KUKA KRL program: sieben_mit.src, sieben_mit.dat

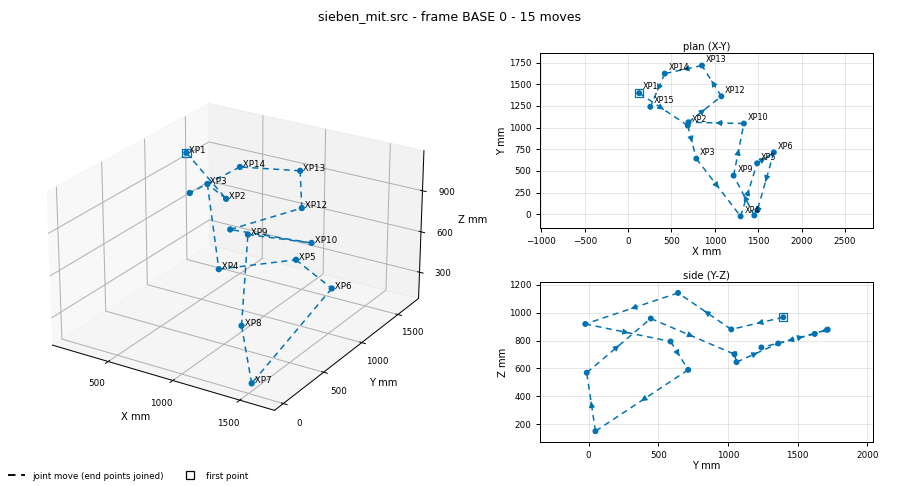
[picture p0: tool path of sieben_mit.src in frame BASE 0, 15 of 17 moves have a stored position in this frame; points joined in program order, loops and branches not executed]
--- sieben_mit.src ---
&ACCESS RVP
&REL 30
&PARAM EDITMASK = *
&PARAM TEMPLATE = C:\KRC\Roboter\Template\vorgabe
DEF sieben_mit( )
;FOLD INI;%{PE}
  ;FOLD BASISTECH INI
    GLOBAL INTERRUPT DECL 3 WHEN $STOPMESS==TRUE DO IR_STOPM ( )
    INTERRUPT ON 3
    BAS (#INITMOV,0 )
  ;ENDFOLD (BASISTECH INI)
  ;FOLD USER INI
    ;Make your modifications here

  ;ENDFOLD (USER INI)
;ENDFOLD (INI)

;FOLD PTP HOME Vel=10 % DEFAULT;%{PE}%R 8.3.40,%MKUKATPBASIS,%CMOVE,%VPTP,%P 1:PTP, 2:HOME, 3:, 5:10, 7:DEFAULT
$BWDSTART=FALSE
PDAT_ACT=PDEFAULT
FDAT_ACT=FHOME
BAS(#PTP_PARAMS,10)
$H_POS=XHOME
PTP XHOME
;ENDFOLD

WAIT FOR IS_KEY_PRESSED(12)

;FOLD PTP P1 Vel=30 % PDAT1 Tool[12]:jan_test Base[0];%{PE}%R 8.3.40,%MKUKATPBASIS,%CMOVE,%VPTP,%P 1:PTP, 2:P1, 3:, 5:30, 7:PDAT1
$BWDSTART=FALSE
PDAT_ACT=PPDAT1
FDAT_ACT=FP1
BAS(#PTP_PARAMS,30)
PTP XP1
;ENDFOLD

WAIT FOR IS_KEY_PRESSED(12)

;FOLD PTP P2 Vel=30 % PDAT2 Tool[12]:jan_test Base[0];%{PE}%R 8.3.40,%MKUKATPBASIS,%CMOVE,%VPTP,%P 1:PTP, 2:P2, 3:, 5:30, 7:PDAT2
$BWDSTART=FALSE
PDAT_ACT=PPDAT2
FDAT_ACT=FP2
BAS(#PTP_PARAMS,30)
PTP XP2
;ENDFOLD

WAIT FOR IS_KEY_PRESSED(12)

;FOLD PTP P3 Vel=30 % PDAT3 Tool[12]:jan_test Base[0];%{PE}%R 8.3.40,%MKUKATPBASIS,%CMOVE,%VPTP,%P 1:PTP, 2:P3, 3:, 5:30, 7:PDAT3
$BWDSTART=FALSE
PDAT_ACT=PPDAT3
FDAT_ACT=FP3
BAS(#PTP_PARAMS,30)
PTP XP3
;ENDFOLD

WAIT FOR IS_KEY_PRESSED(12)

;FOLD PTP P4 Vel=30 % PDAT4 Tool[12]:jan_test Base[0];%{PE}%R 8.3.40,%MKUKATPBASIS,%CMOVE,%VPTP,%P 1:PTP, 2:P4, 3:, 5:30, 7:PDAT4
$BWDSTART=FALSE
PDAT_ACT=PPDAT4
FDAT_ACT=FP4
BAS(#PTP_PARAMS,30)
PTP XP4
;ENDFOLD

WAIT FOR IS_KEY_PRESSED(12)

;FOLD PTP P5 Vel=30 % PDAT5 Tool[12]:jan_test Base[0];%{PE}%R 8.3.40,%MKUKATPBASIS,%CMOVE,%VPTP,%P 1:PTP, 2:P5, 3:, 5:30, 7:PDAT5
$BWDSTART=FALSE
PDAT_ACT=PPDAT5
FDAT_ACT=FP5
BAS(#PTP_PARAMS,30)
PTP XP5
;ENDFOLD

WAIT FOR IS_KEY_PRESSED(12)

;FOLD PTP P6 Vel=30 % PDAT6 Tool[12]:jan_test Base[0];%{PE}%R 8.3.40,%MKUKATPBASIS,%CMOVE,%VPTP,%P 1:PTP, 2:P6, 3:, 5:30, 7:PDAT6
$BWDSTART=FALSE
PDAT_ACT=PPDAT6
FDAT_ACT=FP6
BAS(#PTP_PARAMS,30)
PTP XP6
;ENDFOLD

WAIT FOR IS_KEY_PRESSED(12)

;FOLD PTP P7 Vel=30 % PDAT7 Tool[12]:jan_test Base[0];%{PE}%R 8.3.40,%MKUKATPBASIS,%CMOVE,%VPTP,%P 1:PTP, 2:P7, 3:, 5:30, 7:PDAT7
$BWDSTART=FALSE
PDAT_ACT=PPDAT7
FDAT_ACT=FP7
BAS(#PTP_PARAMS,30)
PTP XP7
;ENDFOLD

WAIT FOR IS_KEY_PRESSED(12)

;FOLD PTP P8 Vel=30 % PDAT8 Tool[12]:jan_test Base[0];%{PE}%R 8.3.40,%MKUKATPBASIS,%CMOVE,%VPTP,%P 1:PTP, 2:P8, 3:, 5:30, 7:PDAT8
$BWDSTART=FALSE
PDAT_ACT=PPDAT8
FDAT_ACT=FP8
BAS(#PTP_PARAMS,30)
PTP XP8
;ENDFOLD

WAIT FOR IS_KEY_PRESSED(12)

;FOLD PTP P9 Vel=30 % PDAT9 Tool[12]:jan_test Base[0];%{PE}%R 8.3.40,%MKUKATPBASIS,%CMOVE,%VPTP,%P 1:PTP, 2:P9, 3:, 5:30, 7:PDAT9
$BWDSTART=FALSE
PDAT_ACT=PPDAT9
FDAT_ACT=FP9
BAS(#PTP_PARAMS,30)
PTP XP9
;ENDFOLD

WAIT FOR IS_KEY_PRESSED(12)

;FOLD PTP P10 Vel=30 % PDAT10 Tool[12]:jan_test Base[0];%{PE}%R 8.3.40,%MKUKATPBASIS,%CMOVE,%VPTP,%P 1:PTP, 2:P10, 3:, 5:30, 7:PDAT10
$BWDSTART=FALSE
PDAT_ACT=PPDAT10
FDAT_ACT=FP10
BAS(#PTP_PARAMS,30)
PTP XP10
;ENDFOLD

WAIT FOR IS_KEY_PRESSED(12)

;FOLD PTP P11 Vel=30 % PDAT11 Tool[12]:jan_test Base[0];%{PE}%R 8.3.40,%MKUKATPBASIS,%CMOVE,%VPTP,%P 1:PTP, 2:P11, 3:, 5:30, 7:PDAT11
$BWDSTART=FALSE
PDAT_ACT=PPDAT11
FDAT_ACT=FP11
BAS(#PTP_PARAMS,30)
PTP XP11
;ENDFOLD

WAIT FOR IS_KEY_PRESSED(12)

;FOLD PTP P12 Vel=30 % PDAT12 Tool[12]:jan_test Base[0];%{PE}%R 8.3.40,%MKUKATPBASIS,%CMOVE,%VPTP,%P 1:PTP, 2:P12, 3:, 5:30, 7:PDAT12
$BWDSTART=FALSE
PDAT_ACT=PPDAT12
FDAT_ACT=FP12
BAS(#PTP_PARAMS,30)
PTP XP12
;ENDFOLD

WAIT FOR IS_KEY_PRESSED(12)

;FOLD PTP P13 Vel=30 % PDAT13 Tool[12]:jan_test Base[0];%{PE}%R 8.3.40,%MKUKATPBASIS,%CMOVE,%VPTP,%P 1:PTP, 2:P13, 3:, 5:30, 7:PDAT13
$BWDSTART=FALSE
PDAT_ACT=PPDAT13
FDAT_ACT=FP13
BAS(#PTP_PARAMS,30)
PTP XP13
;ENDFOLD

WAIT FOR IS_KEY_PRESSED(12)

;FOLD PTP P14 Vel=30 % PDAT14 Tool[12]:jan_test Base[0];%{PE}%R 8.3.40,%MKUKATPBASIS,%CMOVE,%VPTP,%P 1:PTP, 2:P14, 3:, 5:30, 7:PDAT14
$BWDSTART=FALSE
PDAT_ACT=PPDAT14
FDAT_ACT=FP14
BAS(#PTP_PARAMS,30)
PTP XP14
;ENDFOLD

WAIT FOR IS_KEY_PRESSED(12)

;FOLD PTP P15 Vel=30 % PDAT15 Tool[12]:jan_test Base[0];%{PE}%R 8.3.40,%MKUKATPBASIS,%CMOVE,%VPTP,%P 1:PTP, 2:P15, 3:, 5:30, 7:PDAT15
$BWDSTART=FALSE
PDAT_ACT=PPDAT15
FDAT_ACT=FP15
BAS(#PTP_PARAMS,30)
PTP XP15
;ENDFOLD







;FOLD PTP HOME Vel=10 % DEFAULT;%{PE}%R 8.3.40,%MKUKATPBASIS,%CMOVE,%VPTP,%P 1:PTP, 2:HOME, 3:, 5:10, 7:DEFAULT
$BWDSTART=FALSE
PDAT_ACT=PDEFAULT
FDAT_ACT=FHOME
BAS(#PTP_PARAMS,10)
$H_POS=XHOME
PTP XHOME
;ENDFOLD

END

--- sieben_mit.dat ---
&ACCESS RVP
&REL 30
&PARAM EDITMASK = *
&PARAM TEMPLATE = C:\KRC\Roboter\Template\vorgabe
DEFDAT  sieben_mit
;FOLD EXTERNAL DECLARATIONS;%{PE}%MKUKATPBASIS,%CEXT,%VCOMMON,%P
;FOLD BASISTECH EXT;%{PE}%MKUKATPBASIS,%CEXT,%VEXT,%P
EXT  BAS (BAS_COMMAND  :IN,REAL  :IN )
DECL INT SUCCESS
;ENDFOLD (BASISTECH EXT)
;FOLD USER EXT;%{E}%MKUKATPUSER,%CEXT,%VEXT,%P
;Make your modifications here

;ENDFOLD (USER EXT)
;ENDFOLD (EXTERNAL DECLARATIONS)
DECL BASIS_SUGG_T LAST_BASIS={POINT1[] "P15                     ",POINT2[] "P15                     ",CP_PARAMS[] "CPDAT0                  ",PTP_PARAMS[] "PDAT15                  ",CONT[] "                        ",CP_VEL[] "2.0                     ",PTP_VEL[] "30                      ",SYNC_PARAMS[] "SYNCDAT                 ",SPL_NAME[] "S0                      ",A_PARAMS[] "ADAT0                   "}
DECL E6POS XP1={X 127.121788,Y 1397.60730,Z 966.878418,A 28.9919910,B 72.7776489,C -80.1574097,S 18,T 35,E1 0.00499581080,E2 20160.0,E3 0.0,E4 0.0,E5 0.0,E6 0.0}
DECL FDAT FP1={TOOL_NO 12,BASE_NO 0,IPO_FRAME #BASE,POINT2[] " ",TQ_STATE FALSE}
DECL PDAT PPDAT1={VEL 100.000,ACC 50.0000,APO_DIST 100.000,APO_MODE #CDIS,GEAR_JERK 50.0000,EXAX_IGN 0}
DECL E6POS XP2={X 687.482056,Y 1024.24646,Z 879.843384,A 158.221695,B 27.4421253,C 130.372269,S 18,T 35,E1 0.00499581080,E2 20160.0,E3 0.0,E4 0.0,E5 0.0,E6 0.0}
DECL FDAT FP2={TOOL_NO 12,BASE_NO 0,IPO_FRAME #BASE,POINT2[] " ",TQ_STATE FALSE}
DECL PDAT PPDAT2={VEL 100.000,ACC 50.0000,APO_DIST 100.000,APO_MODE #CDIS,GEAR_JERK 50.0000,EXAX_IGN 0}
DECL E6POS XP3={X 786.710938,Y 642.340820,Z 1141.43823,A -17.2900,B 75.0733795,C -84.1357117,S 18,T 35,E1 0.00499581080,E2 20160.0,E3 0.0,E4 0.0,E5 0.0,E6 0.0}
DECL FDAT FP3={TOOL_NO 12,BASE_NO 0,IPO_FRAME #BASE,POINT2[] " ",TQ_STATE FALSE}
DECL PDAT PPDAT3={VEL 100.000,ACC 50.0000,APO_DIST 100.000,APO_MODE #CDIS,GEAR_JERK 50.0000,EXAX_IGN 0}
DECL E6POS XP4={X 1297.19812,Y -23.5658340,Z 918.717651,A 143.866684,B 43.7865524,C 154.133148,S 18,T 34,E1 0.00499581080,E2 20160.0,E3 0.0,E4 0.0,E5 0.0,E6 0.0}
DECL FDAT FP4={TOOL_NO 12,BASE_NO 0,IPO_FRAME #BASE,POINT2[] " ",TQ_STATE FALSE}
DECL PDAT PPDAT4={VEL 100.000,ACC 50.0000,APO_DIST 100.000,APO_MODE #CDIS,GEAR_JERK 50.0000,EXAX_IGN 0}
DECL E6POS XP5={X 1487.88892,Y 588.539063,Z 793.160034,A 169.410522,B 66.9371109,C 101.298386,S 18,T 35,E1 0.00499581080,E2 20160.0,E3 0.0,E4 0.0,E5 0.0,E6 0.0}
DECL FDAT FP5={TOOL_NO 12,BASE_NO 0,IPO_FRAME #BASE,POINT2[] " ",TQ_STATE FALSE}
DECL PDAT PPDAT5={VEL 100.000,ACC 50.0000,APO_DIST 100.000,APO_MODE #CDIS,GEAR_JERK 50.0000,EXAX_IGN 0}
DECL E6POS XP6={X 1680.46313,Y 714.720581,Z 589.578308,A -139.295685,B 53.2188530,C -171.760605,S 18,T 35,E1 0.00499581080,E2 20160.0,E3 0.0,E4 0.0,E5 0.0,E6 0.0}
DECL FDAT FP6={TOOL_NO 12,BASE_NO 0,IPO_FRAME #BASE,POINT2[] " ",TQ_STATE FALSE}
DECL PDAT PPDAT6={VEL 100.000,ACC 50.0000,APO_DIST 100.000,APO_MODE #CDIS,GEAR_JERK 50.0000,EXAX_IGN 0}
DECL E6POS XP7={X 1491.72949,Y 49.5089493,Z 149.166748,A 178.390442,B -4.23892879,C -161.530624,S 22,T 51,E1 0.00499581080,E2 20160.0,E3 0.0,E4 0.0,E5 0.0,E6 0.0}
DECL FDAT FP7={TOOL_NO 12,BASE_NO 0,IPO_FRAME #BASE,POINT2[] " ",TQ_STATE FALSE}
DECL PDAT PPDAT7={VEL 100.000,ACC 50.0000,APO_DIST 100.000,APO_MODE #CDIS,GEAR_JERK 50.0000,EXAX_IGN 0}
DECL E6POS XP8={X 1455.62463,Y -13.2068548,Z 568.786499,A -137.534805,B 55.8855133,C 177.677444,S 18,T 34,E1 0.00499581080,E2 20160.0,E3 0.0,E4 0.0,E5 0.0,E6 0.0}
DECL FDAT FP8={TOOL_NO 12,BASE_NO 0,IPO_FRAME #BASE,POINT2[] " ",TQ_STATE FALSE}
DECL PDAT PPDAT8={VEL 100.000,ACC 50.0000,APO_DIST 100.000,APO_MODE #CDIS,GEAR_JERK 50.0000,EXAX_IGN 0}
DECL E6POS XP9={X 1216.24670,Y 446.606415,Z 957.778320,A 140.879868,B 69.8143,C 45.8475914,S 18,T 35,E1 0.00499581080,E2 20160.0,E3 0.0,E4 0.0,E5 0.0,E6 0.0}
DECL FDAT FP9={TOOL_NO 12,BASE_NO 0,IPO_FRAME #BASE,POINT2[] " ",TQ_STATE FALSE}
DECL PDAT PPDAT9={VEL 100.000,ACC 50.0000,APO_DIST 100.000,APO_MODE #CDIS,GEAR_JERK 50.0000,EXAX_IGN 0}
DECL E6POS XP10={X 1335.25195,Y 1047.45752,Z 701.586426,A -66.7826538,B 76.0818710,C -128.477203,S 18,T 35,E1 0.00499581080,E2 20160.0,E3 0.0,E4 0.0,E5 0.0,E6 0.0}
DECL FDAT FP10={TOOL_NO 12,BASE_NO 0,IPO_FRAME #BASE,POINT2[] " ",TQ_STATE FALSE}
DECL PDAT PPDAT10={VEL 100.000,ACC 50.0000,APO_DIST 100.000,APO_MODE #CDIS,GEAR_JERK 50.0000,EXAX_IGN 0}
DECL E6POS XP11={X 695.521790,Y 1061.91431,Z 644.949280,A -126.047440,B 67.4937057,C 104.088135,S 18,T 35,E1 0.00503292447,E2 20160.0,E3 0.0,E4 0.0,E5 0.0,E6 0.0}
DECL FDAT FP11={TOOL_NO 12,BASE_NO 0,IPO_FRAME #BASE,POINT2[] " ",TQ_STATE FALSE}
DECL PDAT PPDAT11={VEL 100.000,ACC 50.0000,APO_DIST 100.000,APO_MODE #CDIS,GEAR_JERK 50.0000,EXAX_IGN 0}
DECL E6POS XP12={X 1075.02905,Y 1361.14771,Z 778.891479,A 163.397339,B 34.7752914,C 85.8660278,S 18,T 35,E1 0.00505519472,E2 20160.0,E3 0.0,E4 0.0,E5 0.0,E6 0.0}
DECL FDAT FP12={TOOL_NO 12,BASE_NO 0,IPO_FRAME #BASE,POINT2[] " ",TQ_STATE FALSE}
DECL PDAT PPDAT12={VEL 100.000,ACC 50.0000,APO_DIST 100.000,APO_MODE #CDIS,GEAR_JERK 50.0000,EXAX_IGN 0}
DECL E6POS XP13={X 851.128845,Y 1716.49036,Z 878.567810,A 138.041687,B -23.8696175,C 120.093315,S 18,T 35,E1 0.00505519472,E2 20160.0,E3 0.0,E4 0.0,E5 0.0,E6 0.0}
DECL FDAT FP13={TOOL_NO 12,BASE_NO 0,IPO_FRAME #BASE,POINT2[] " ",TQ_STATE FALSE}
DECL PDAT PPDAT13={VEL 100.000,ACC 50.0000,APO_DIST 100.000,APO_MODE #CDIS,GEAR_JERK 50.0000,EXAX_IGN 0}
DECL E6POS XP14={X 421.905396,Y 1623.28625,Z 847.276611,A -156.940399,B 79.2187119,C 136.989288,S 18,T 35,E1 0.00505519472,E2 20160.0,E3 0.0,E4 0.0,E5 0.0,E6 0.0}
DECL FDAT FP14={TOOL_NO 12,BASE_NO 0,IPO_FRAME #BASE,POINT2[] " ",TQ_STATE FALSE}
DECL PDAT PPDAT14={VEL 100.000,ACC 50.0000,APO_DIST 100.000,APO_MODE #CDIS,GEAR_JERK 50.0000,EXAX_IGN 0}
DECL E6POS XP15={X 255.608322,Y 1240.22705,Z 750.276794,A 132.350601,B 87.8609085,C 64.6111450,S 18,T 35,E1 0.00521850819,E2 20160.0,E3 0.0,E4 0.0,E5 0.0,E6 0.0}
DECL FDAT FP15={TOOL_NO 12,BASE_NO 0,IPO_FRAME #BASE,POINT2[] " ",TQ_STATE FALSE}
DECL PDAT PPDAT15={VEL 100.000,ACC 50.0000,APO_DIST 100.000,APO_MODE #CDIS,GEAR_JERK 50.0000,EXAX_IGN 0}
ENDDAT
